TEXTLIST AnyStationAlarmList
  0 = ' '
  1 = 'Station 1 Fault'
  2 = 'Station 2 Fault'
  3 = 'Station 3 Fault'
  4 = 'Station 4 Fault'
  5 = 'Station 5 Fault'
  6 = 'Station 6 Fault'
  99 = 'Machine Fault'
   = ''
END_TEXTLIST

(* stored: Version 1.1.0.1, ProductVersion 3.1.4024.12
   TextList AnyStationAlarmList: Id {a439557a-ee7b-47b6-a50d-7bdfc2489f71} *)
